// SIMATIC S7-200 project (STEP 7-Micro/WIN), CPU 224XP CN REL 02.01

ORGANIZATION_BLOCK 程序块:OB1
TITLE=该程序通过S7-200 PLC利用Modbus主站库与LG变频器进行通讯，实现对电机的远程控制，用于精确控制电机转速。
// 系统启动时，系统始终使能标志驱动Modbus控制初始化功能。
// 当操作员按下正向启动按钮，且反向启动按钮和停止按钮未按下时，正向运行标志置位，防止正反向命令冲突。
// 随即，设置电机转速设定值为正向运行命令，并准备Modbus寄存器地址，正向启动延时定时器计时后复位标志，确保启动过程平稳完成。
// 随后，通过Modbus消息发送功能将数据写入变频器。
// 反向启动按钮按下时，若正向启动按钮和停止按钮未激活，反向运行标志置位。
// 随即，在系统特定状态下，设置电机转速设定值为反向运行命令，并准备Modbus寄存器地址，反向启动延时定时器计时后复位，避免运行状态混乱。
// 若操作员按下停止按钮，且反向启动按钮和其他条件未激活，停止运行标志置位。
// 随即，在系统特定状态下，设置电机转速设定值为0，并准备Modbus寄存器地址，停止延时定时器计时后复位，确保传送带完全停止。
// 转速调整通过设置电机转速设定值，并从电机当前转速值实时反馈。
// 随后，在Modbus通信正常运行时，通过Modbus消息发送功能将数据写入变频器。
// 这个程序是利用Modbus指令库做的，这种指令库目前没有太多资料。不能完全按库上面的注解来做，不然死的惨。我是用串口工具才调试出来的，在这个网站拿了不少东西。今天我也贡献一点点，希望网站上资料会越来越多。
BEGIN
Network 1 // Network Title
// Network Comment
LD     SM0.0
=      L60.0
LD     SM0.0
=      L63.7
LD     L60.0
CALL   MBUS_CTRL:SBR1, L63.7, 19200, 0, 1000, M20.2, VB502
Network 2
LD     T36
=      M2.6
S      M2.7, 1
Network 3
LDN    M2.3
AN     M2.1
AN     M2.2
MOVW   VW680, VW660
MOVD   40006, VD602
Network 4
LD     SM0.0
=      L60.0
LD     SM0.0
=      L63.7
LD     L60.0
CALL   MBUS_MSG:SBR2, L63.7, 1, 1, VD602, 1, &VB600, M20.1, VB506
Network 6
LD     SM0.0
MOVW   VW660, VW600
Network 7
// 正向起动
LD     M20.6
AN     M21.1
AN     M21.2
EU
S      M2.1, 1
Network 8
// 正向起动
LD     M2.1
LPS
MOVW   16#2, VW660
MOVD   40007, VD602
TON    T33, 200
ED
TOF    T36, 500
LPP
A      T33
R      M2.1, 1
Network 9
// 反向起动
LD     M21.1
AN     M20.6
AN     M21.2
EU
S      M2.2, 1
Network 10
// 反向起动
LD     M2.2
LPS
AN     SM0.5
MOVW   16#4, VW660
LRD
AN     SM0.5
MOVD   40007, VD602
LRD
TON    T34, 200
LPP
A      T34
R      M2.2, 1
Network 11
// 停止
LD     M21.2
AN     M21.1
AN     M21.6
EU
S      M2.3, 1
Network 12
// 停止
LD     M2.3
LPS
AN     SM0.5
MOVW   16#0, VW660
LRD
AN     SM0.5
MOVD   40007, VD602
LRD
TON    T35, 300
LPP
A      T35
R      M2.3, 1
END_ORGANIZATION_BLOCK

// SBR1: protected block, not included

// SBR2: protected block, not included

// SBR3: protected block, not included
